// TIA Portal V20 export
TYPE "typeCmControlNodeSoftCam"
// stored: Namespace Unit1.Em6
   STRUCT
      visionUnit { ExternalWritable := 'False'} : "Unit1.Em6.typeCmControlNodeSoftCamVisionController";
   END_STRUCT;
END_TYPE
